// Mitsubishi GX Works2 project: Fx1NC-32MT-getfromInit   PLC: FX1N/FX1NC

PROGRAM MAIN
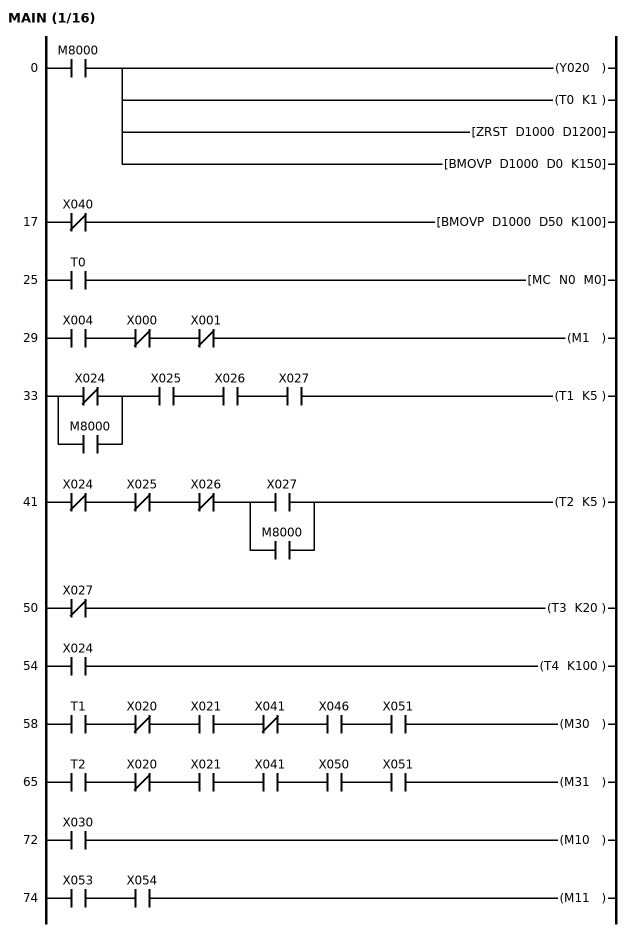
0     LD      M8000
      OUT     Y020
      OUT     T0 K1
      ZRST    D1000 D1200
      BMOVP   D1000 D0 K150
17    LDI     X040
      BMOVP   D1000 D50 K100
25    LD      T0
      MC      N0 M0
29    LD      X004
      ANI     X000
      ANI     X001
      OUT     M1
33    LDI     X024
      OR      M8000
      AND     X025
      AND     X026
      AND     X027
      OUT     T1 K5
41    LDI     X024
      ANI     X025
      ANI     X026
      LD      X027
      OR      M8000
      ANB
      OUT     T2 K5
50    LDI     X027
      OUT     T3 K20
54    LD      X024
      OUT     T4 K100
58    LD      T1
      ANI     X020
      AND     X021
      ANI     X041
      AND     X046
      AND     X051
      OUT     M30
65    LD      T2
      ANI     X020
      AND     X021
      AND     X041
      AND     X050
      AND     X051
      OUT     M31
72    LD      X030
      OUT     M10
74    LD      X053
      AND     X054
      OUT     M11
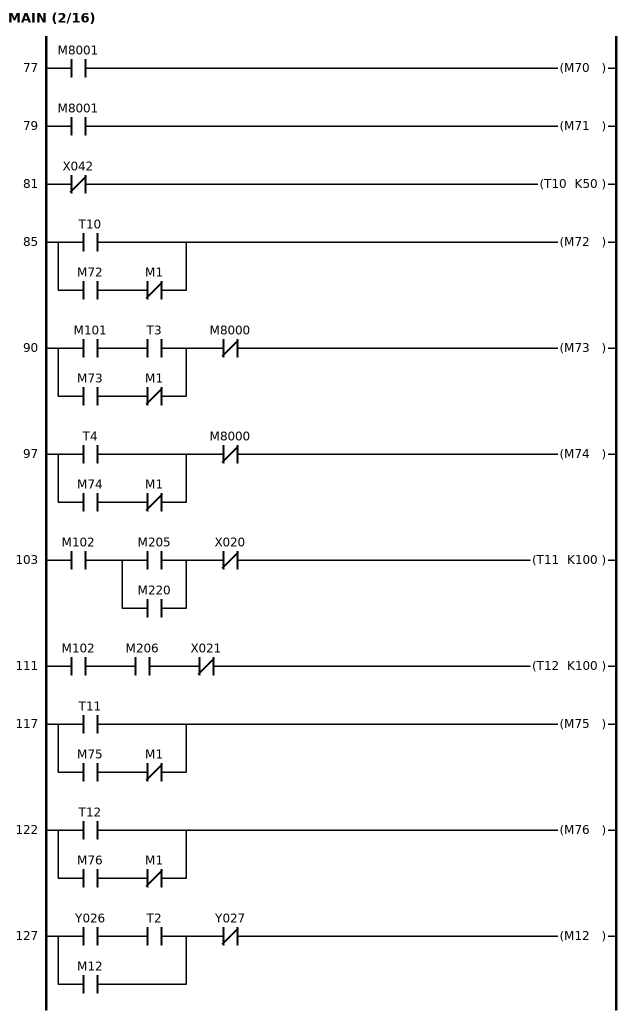
77    LD      M8001
      OUT     M70
79    LD      M8001
      OUT     M71
81    LDI     X042
      OUT     T10 K50
85    LD      T10
      LD      M72
      ANI     M1
      ORB
      OUT     M72
90    LD      M101
      AND     T3
      LD      M73
      ANI     M1
      ORB
      ANI     M8000
      OUT     M73
97    LD      T4
      LD      M74
      ANI     M1
      ORB
      ANI     M8000
      OUT     M74
103   LD      M102
      LD      M205
      OR      M220
      ANB
      ANI     X020
      OUT     T11 K100
111   LD      M102
      AND     M206
      ANI     X021
      OUT     T12 K100
117   LD      T11
      LD      M75
      ANI     M1
      ORB
      OUT     M75
122   LD      T12
      LD      M76
      ANI     M1
      ORB
      OUT     M76
127   LD      Y026
      AND     T2
      OR      M12
      ANI     Y027
      OUT     M12
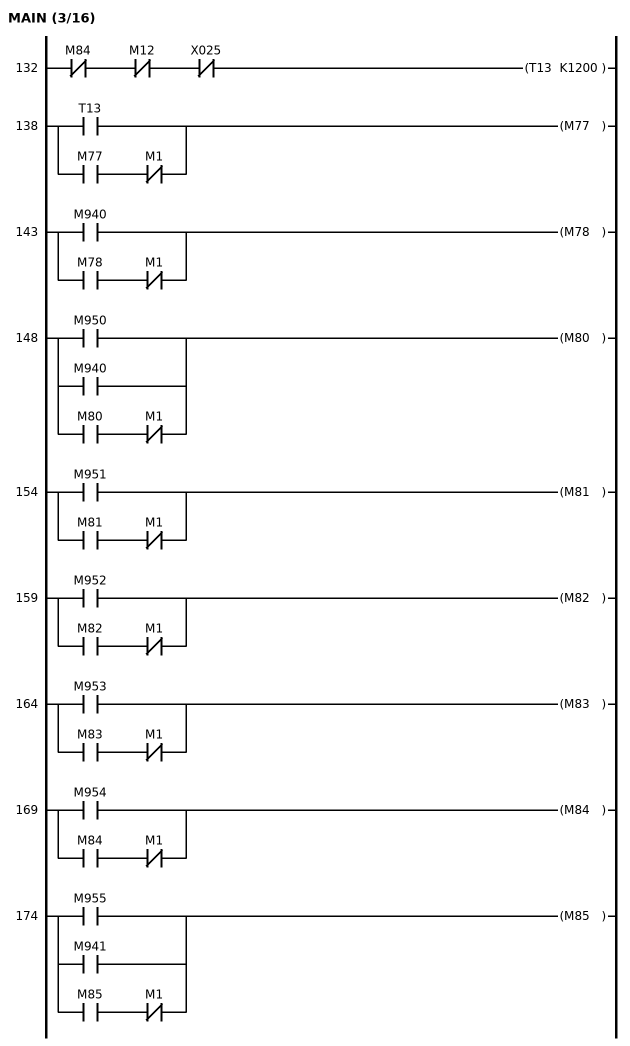
132   LDI     M84
      ANI     M12
      ANI     X025
      OUT     T13 K1200
138   LD      T13
      LD      M77
      ANI     M1
      ORB
      OUT     M77
143   LD      M940
      LD      M78
      ANI     M1
      ORB
      OUT     M78
148   LD      M950
      OR      M940
      LD      M80
      ANI     M1
      ORB
      OUT     M80
154   LD      M951
      LD      M81
      ANI     M1
      ORB
      OUT     M81
159   LD      M952
      LD      M82
      ANI     M1
      ORB
      OUT     M82
164   LD      M953
      LD      M83
      ANI     M1
      ORB
      OUT     M83
169   LD      M954
      LD      M84
      ANI     M1
      ORB
      OUT     M84
174   LD      M955
      OR      M941
      LD      M85
      ANI     M1
      ORB
      OUT     M85
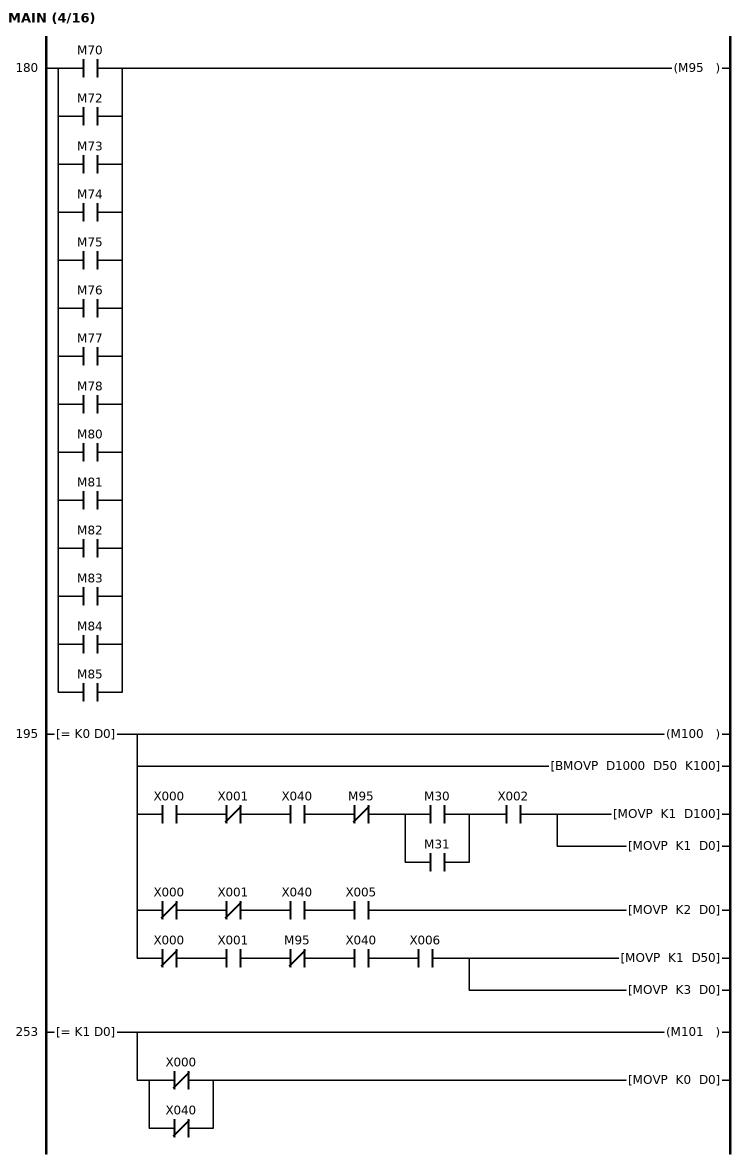
180   LD      M70
      OR      M72
      OR      M73
      OR      M74
      OR      M75
      OR      M76
      OR      M77
      OR      M78
      OR      M80
      OR      M81
      OR      M82
      OR      M83
      OR      M84
      OR      M85
      OUT     M95
195   LD=     K0 D0
      OUT     M100
      BMOVP   D1000 D50 K100
      MPS
      AND     X000
      ANI     X001
      AND     X040
      ANI     M95
      LD      M30
      OR      M31
      ANB
      AND     X002
      MOVP    K1 D100
      MOVP    K1 D0
      MRD
      ANI     X000
      ANI     X001
      AND     X040
      AND     X005
      MOVP    K2 D0
      MPP
      ANI     X000
      AND     X001
      ANI     M95
      AND     X040
      AND     X006
      MOVP    K1 D50
      MOVP    K3 D0
253   LD=     K1 D0
      OUT     M101
      LDI     X000
      ORI     X040
      ANB
      MOVP    K0 D0
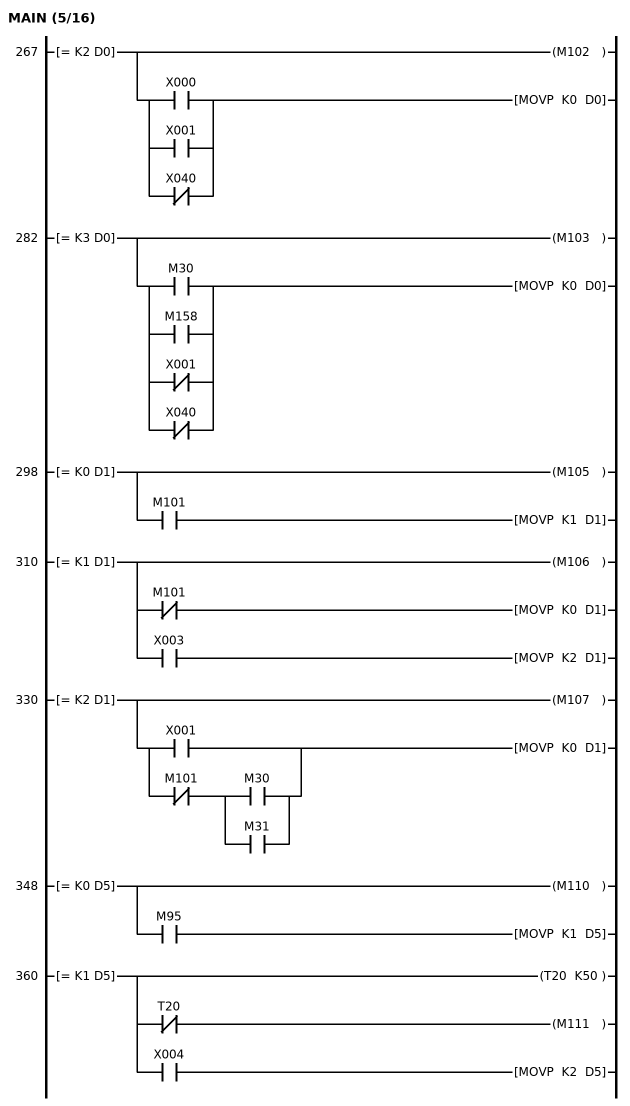
267   LD=     K2 D0
      OUT     M102
      LD      X000
      OR      X001
      ORI     X040
      ANB
      MOVP    K0 D0
282   LD=     K3 D0
      OUT     M103
      LD      M30
      OR      M158
      ORI     X001
      ORI     X040
      ANB
      MOVP    K0 D0
298   LD=     K0 D1
      OUT     M105
      AND     M101
      MOVP    K1 D1
310   LD=     K1 D1
      OUT     M106
      MPS
      ANI     M101
      MOVP    K0 D1
      MPP
      AND     X003
      MOVP    K2 D1
330   LD=     K2 D1
      OUT     M107
      LD      X001
      LDI     M101
      LD      M30
      OR      M31
      ANB
      ORB
      ANB
      MOVP    K0 D1
348   LD=     K0 D5
      OUT     M110
      AND     M95
      MOVP    K1 D5
360   LD=     K1 D5
      OUT     T20 K50
      MPS
      ANI     T20
      OUT     M111
      MPP
      AND     X004
      MOVP    K2 D5
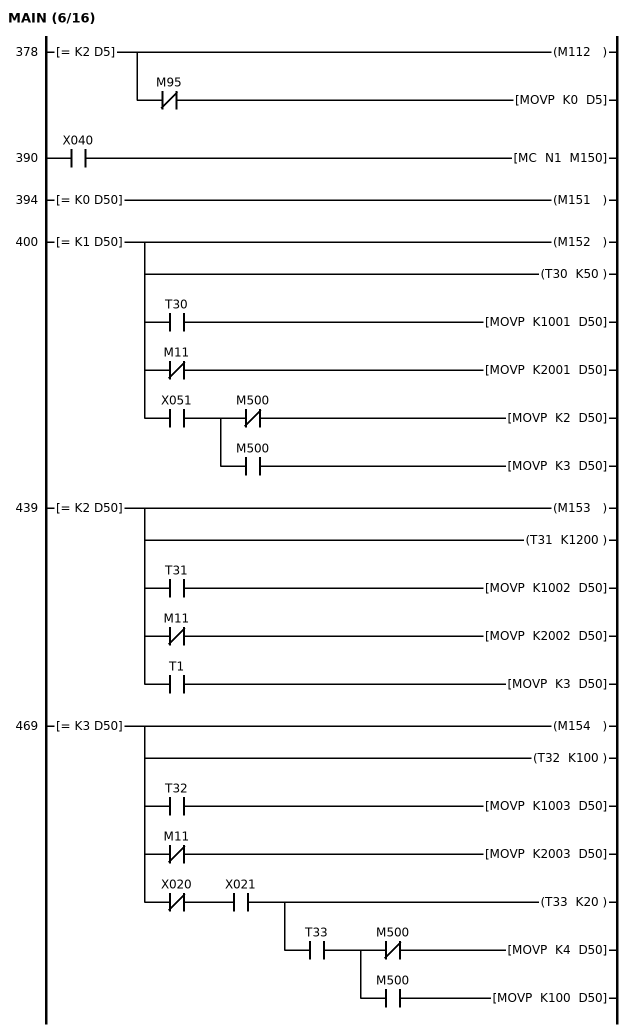
378   LD=     K2 D5
      OUT     M112
      ANI     M95
      MOVP    K0 D5
390   LD      X040
      MC      N1 M150
394   LD=     K0 D50
      OUT     M151
400   LD=     K1 D50
      OUT     M152
      OUT     T30 K50
      MPS
      AND     T30
      MOVP    K1001 D50
      MRD
      ANI     M11
      MOVP    K2001 D50
      MPP
      AND     X051
      MPS
      ANI     M500
      MOVP    K2 D50
      MPP
      AND     M500
      MOVP    K3 D50
439   LD=     K2 D50
      OUT     M153
      OUT     T31 K1200
      MPS
      AND     T31
      MOVP    K1002 D50
      MRD
      ANI     M11
      MOVP    K2002 D50
      MPP
      AND     T1
      MOVP    K3 D50
469   LD=     K3 D50
      OUT     M154
      OUT     T32 K100
      MPS
      AND     T32
      MOVP    K1003 D50
      MRD
      ANI     M11
      MOVP    K2003 D50
      MPP
      ANI     X020
      AND     X021
      OUT     T33 K20
      AND     T33
      MPS
      ANI     M500
      MOVP    K4 D50
      MPP
      AND     M500
      MOVP    K100 D50
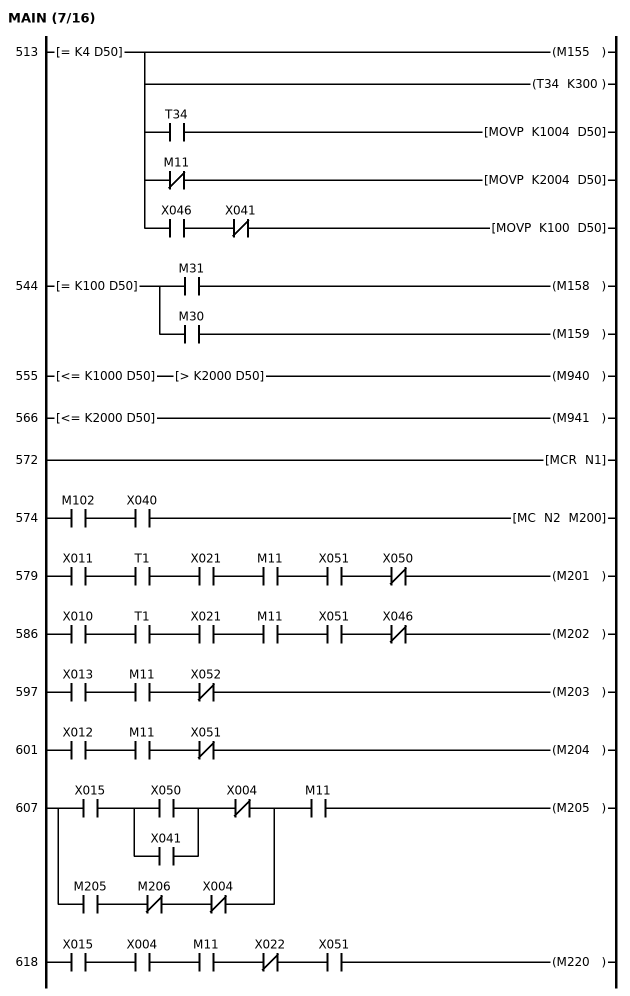
513   LD=     K4 D50
      OUT     M155
      OUT     T34 K300
      MPS
      AND     T34
      MOVP    K1004 D50
      MRD
      ANI     M11
      MOVP    K2004 D50
      MPP
      AND     X046
      ANI     X041
      MOVP    K100 D50
544   LD=     K100 D50
      MPS
      AND     M31
      OUT     M158
      MPP
      AND     M30
      OUT     M159
555   LD<=    K1000 D50
      AND>    K2000 D50
      OUT     M940
566   LD<=    K2000 D50
      OUT     M941
572   MCR     N1
574   LD      M102
      AND     X040
      MC      N2 M200
579   LD      X011
      AND     T1
      AND     X021
      AND     M11
      AND     X051
      ANI     X050
      OUT     M201
586   LD      X010
      AND     T1
      AND     X021
      AND     M11
      AND     X051
      ANI     X046
      OUT     M202
597   LD      X013
      AND     M11
      ANI     X052
      OUT     M203
601   LD      X012
      AND     M11
      ANI     X051
      OUT     M204
607   LD      X015
      LD      X050
      OR      X041
      ANB
      ANI     X004
      LD      M205
      ANI     M206
      ANI     X004
      ORB
      AND     M11
      OUT     M205
618   LD      X015
      AND     X004
      AND     M11
      ANI     X022
      AND     X051
      OUT     M220
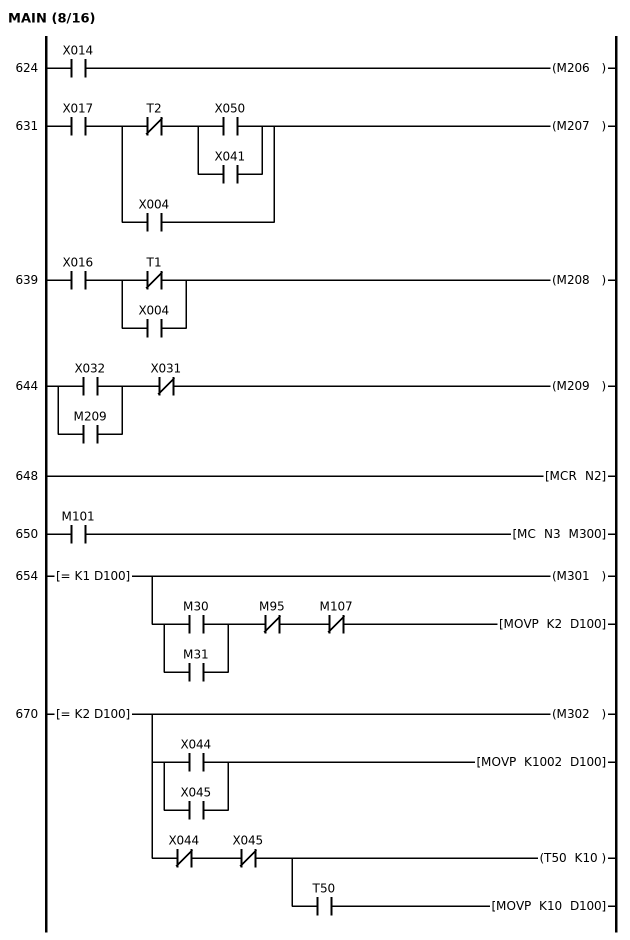
624   LD      X014
      OUT     M206
631   LD      X017
      LDI     T2
      LD      X050
      OR      X041
      ANB
      OR      X004
      ANB
      OUT     M207
639   LD      X016
      LDI     T1
      OR      X004
      ANB
      OUT     M208
644   LD      X032
      OR      M209
      ANI     X031
      OUT     M209
648   MCR     N2
650   LD      M101
      MC      N3 M300
654   LD=     K1 D100
      OUT     M301
      LD      M30
      OR      M31
      ANB
      ANI     M95
      ANI     M107
      MOVP    K2 D100
670   LD=     K2 D100
      OUT     M302
      MPS
      LD      X044
      OR      X045
      ANB
      MOVP    K1002 D100
      MPP
      ANI     X044
      ANI     X045
      OUT     T50 K10
      AND     T50
      MOVP    K10 D100
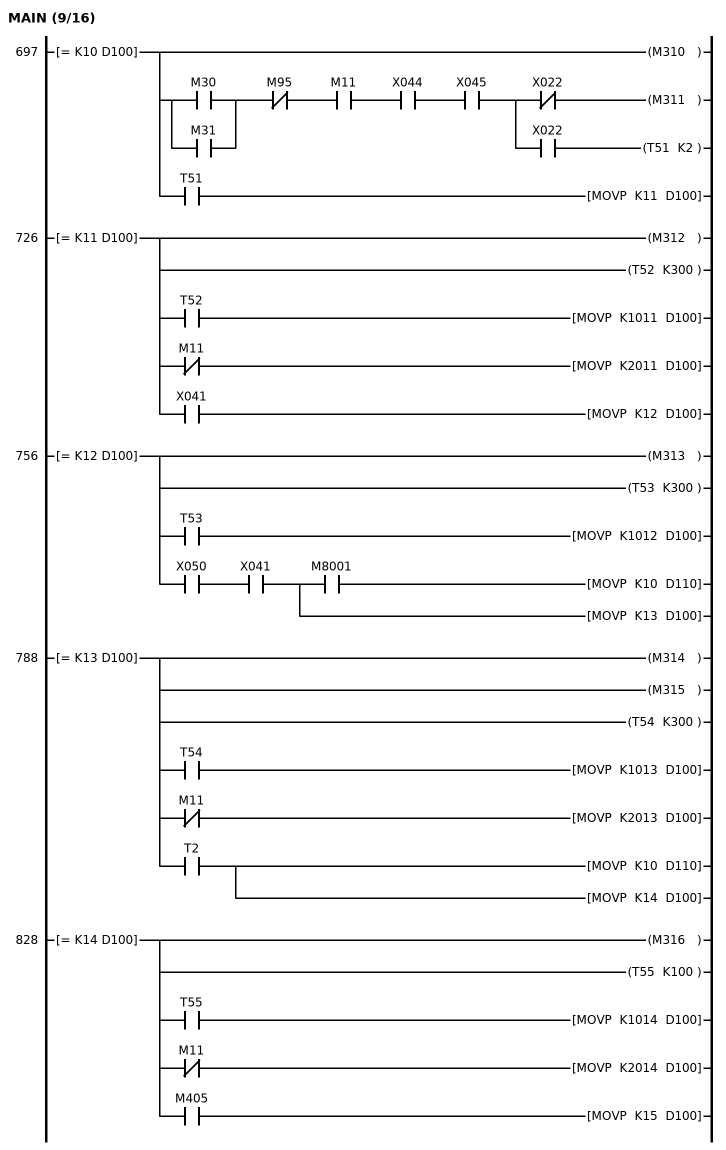
697   LD=     K10 D100
      OUT     M310
      MPS
      LD      M30
      OR      M31
      ANB
      ANI     M95
      AND     M11
      AND     X044
      AND     X045
      MPS
      ANI     X022
      OUT     M311
      MPP
      AND     X022
      OUT     T51 K2
      MPP
      AND     T51
      MOVP    K11 D100
726   LD=     K11 D100
      OUT     M312
      OUT     T52 K300
      MPS
      AND     T52
      MOVP    K1011 D100
      MRD
      ANI     M11
      MOVP    K2011 D100
      MPP
      AND     X041
      MOVP    K12 D100
756   LD=     K12 D100
      OUT     M313
      OUT     T53 K300
      MPS
      AND     T53
      MOVP    K1012 D100
      MPP
      AND     X050
      AND     X041
      MPS
      AND     M8001
      MOVP    K10 D110
      MPP
      MOVP    K13 D100
788   LD=     K13 D100
      OUT     M314
      OUT     M315
      OUT     T54 K300
      MPS
      AND     T54
      MOVP    K1013 D100
      MRD
      ANI     M11
      MOVP    K2013 D100
      MPP
      AND     T2
      MOVP    K10 D110
      MOVP    K14 D100
828   LD=     K14 D100
      OUT     M316
      OUT     T55 K100
      MPS
      AND     T55
      MOVP    K1014 D100
      MRD
      ANI     M11
      MOVP    K2014 D100
      MPP
      AND     M405
      MOVP    K15 D100
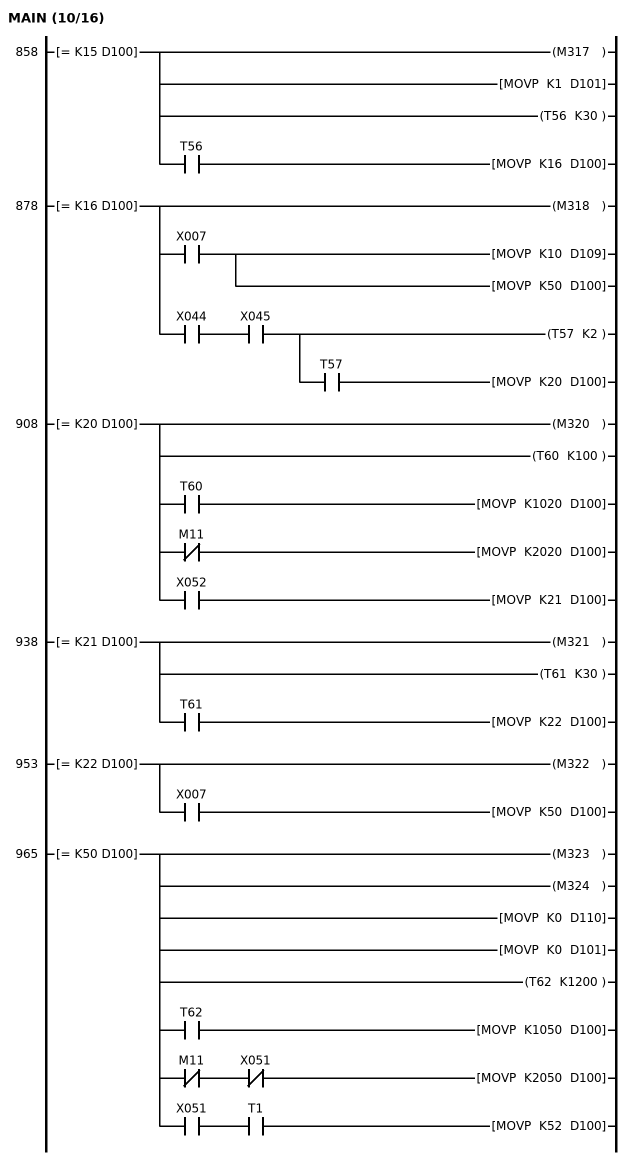
858   LD=     K15 D100
      OUT     M317
      MOVP    K1 D101
      OUT     T56 K30
      AND     T56
      MOVP    K16 D100
878   LD=     K16 D100
      OUT     M318
      MPS
      AND     X007
      MOVP    K10 D109
      MOVP    K50 D100
      MPP
      AND     X044
      AND     X045
      OUT     T57 K2
      AND     T57
      MOVP    K20 D100
908   LD=     K20 D100
      OUT     M320
      OUT     T60 K100
      MPS
      AND     T60
      MOVP    K1020 D100
      MRD
      ANI     M11
      MOVP    K2020 D100
      MPP
      AND     X052
      MOVP    K21 D100
938   LD=     K21 D100
      OUT     M321
      OUT     T61 K30
      AND     T61
      MOVP    K22 D100
953   LD=     K22 D100
      OUT     M322
      AND     X007
      MOVP    K50 D100
965   LD=     K50 D100
      OUT     M323
      OUT     M324
      MOVP    K0 D110
      MOVP    K0 D101
      OUT     T62 K1200
      MPS
      AND     T62
      MOVP    K1050 D100
      MRD
      ANI     M11
      ANI     X051
      MOVP    K2050 D100
      MPP
      AND     X051
      AND     T1
      MOVP    K52 D100
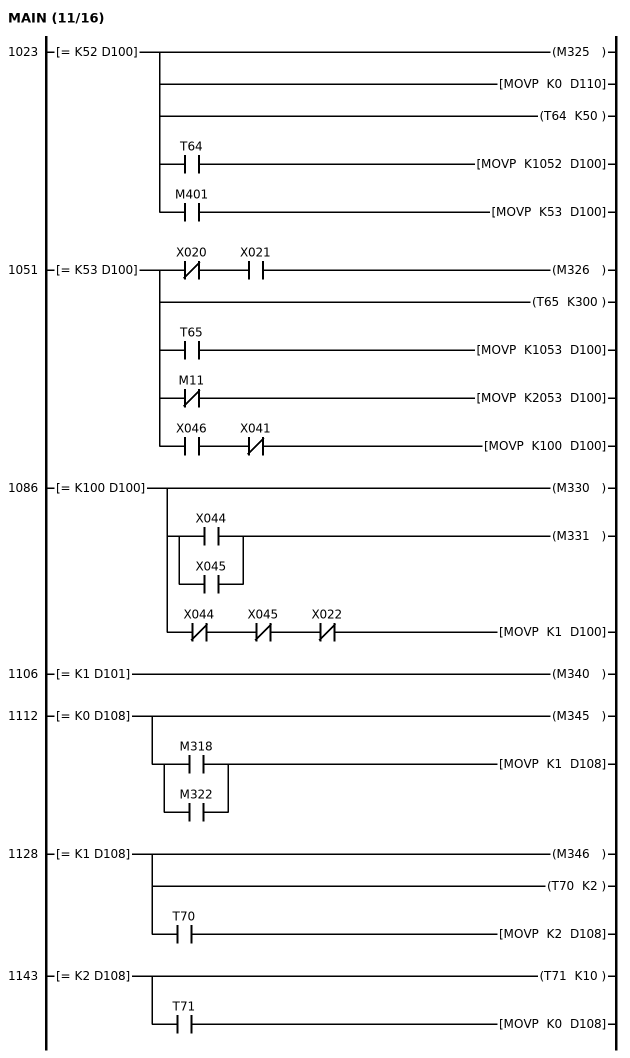
1023  LD=     K52 D100
      OUT     M325
      MOVP    K0 D110
      OUT     T64 K50
      MPS
      AND     T64
      MOVP    K1052 D100
      MPP
      AND     M401
      MOVP    K53 D100
1051  LD=     K53 D100
      MPS
      ANI     X020
      AND     X021
      OUT     M326
      MPP
      OUT     T65 K300
      MPS
      AND     T65
      MOVP    K1053 D100
      MRD
      ANI     M11
      MOVP    K2053 D100
      MPP
      AND     X046
      ANI     X041
      MOVP    K100 D100
1086  LD=     K100 D100
      OUT     M330
      MPS
      LD      X044
      OR      X045
      ANB
      OUT     M331
      MPP
      ANI     X044
      ANI     X045
      ANI     X022
      MOVP    K1 D100
1106  LD=     K1 D101
      OUT     M340
1112  LD=     K0 D108
      OUT     M345
      LD      M318
      OR      M322
      ANB
      MOVP    K1 D108
1128  LD=     K1 D108
      OUT     M346
      OUT     T70 K2
      AND     T70
      MOVP    K2 D108
1143  LD=     K2 D108
      OUT     T71 K10
      AND     T71
      MOVP    K0 D108
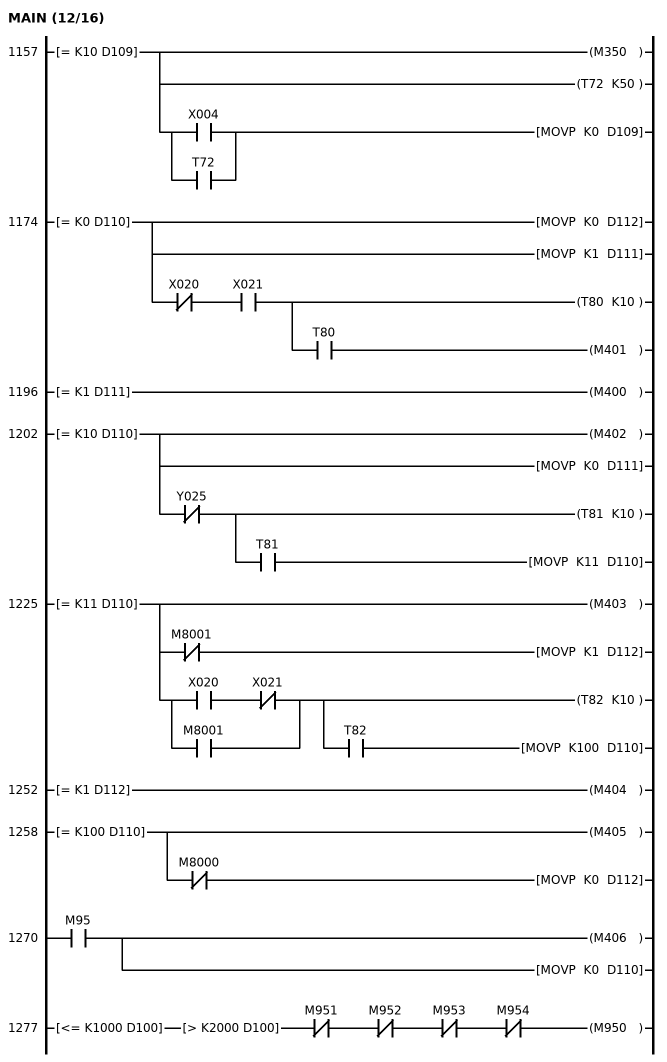
1157  LD=     K10 D109
      OUT     M350
      OUT     T72 K50
      LD      X004
      OR      T72
      ANB
      MOVP    K0 D109
1174  LD=     K0 D110
      MOVP    K0 D112
      MOVP    K1 D111
      ANI     X020
      AND     X021
      OUT     T80 K10
      AND     T80
      OUT     M401
1196  LD=     K1 D111
      OUT     M400
1202  LD=     K10 D110
      OUT     M402
      MOVP    K0 D111
      ANI     Y025
      OUT     T81 K10
      AND     T81
      MOVP    K11 D110
1225  LD=     K11 D110
      OUT     M403
      MPS
      ANI     M8001
      MOVP    K1 D112
      MPP
      LD      X020
      ANI     X021
      OR      M8001
      ANB
      OUT     T82 K10
      AND     T82
      MOVP    K100 D110
1252  LD=     K1 D112
      OUT     M404
1258  LD=     K100 D110
      OUT     M405
      ANI     M8000
      MOVP    K0 D112
1270  LD      M95
      OUT     M406
      MOVP    K0 D110
1277  LD<=    K1000 D100
      AND>    K2000 D100
      ANI     M951
      ANI     M952
      ANI     M953
      ANI     M954
      OUT     M950
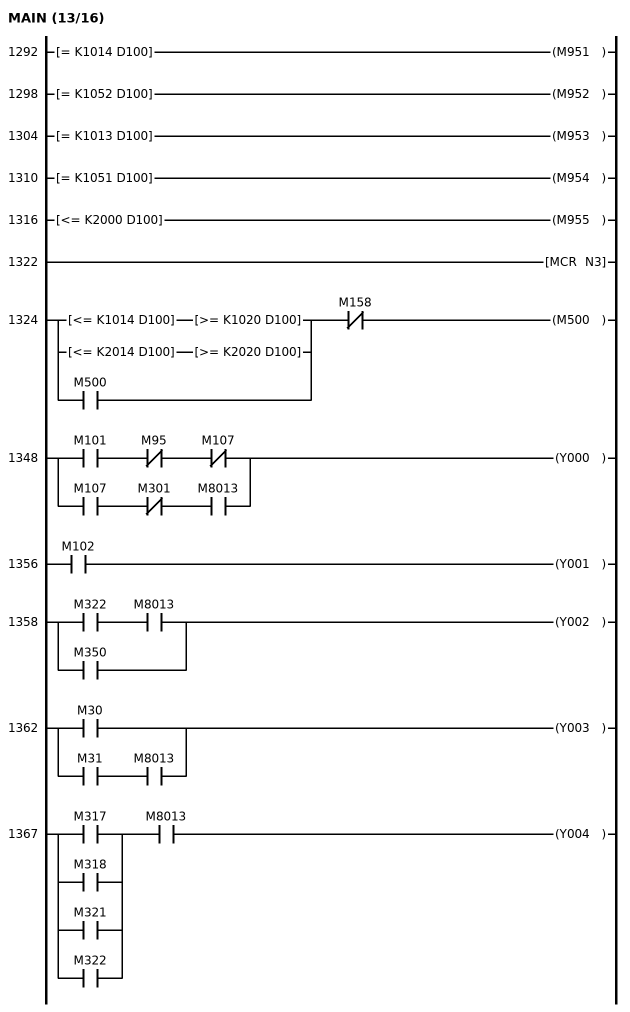
1292  LD=     K1014 D100
      OUT     M951
1298  LD=     K1052 D100
      OUT     M952
1304  LD=     K1013 D100
      OUT     M953
1310  LD=     K1051 D100
      OUT     M954
1316  LD<=    K2000 D100
      OUT     M955
1322  MCR     N3
1324  LD<=    K1014 D100
      AND>=   K1020 D100
      LD<=    K2014 D100
      AND>=   K2020 D100
      ORB
      OR      M500
      ANI     M158
      OUT     M500
1348  LD      M101
      ANI     M95
      ANI     M107
      LD      M107
      ANI     M301
      AND     M8013
      ORB
      OUT     Y000
1356  LD      M102
      OUT     Y001
1358  LD      M322
      AND     M8013
      OR      M350
      OUT     Y002
1362  LD      M30
      LD      M31
      AND     M8013
      ORB
      OUT     Y003
1367  LD      M317
      OR      M318
      OR      M321
      OR      M322
      AND     M8013
      OUT     Y004
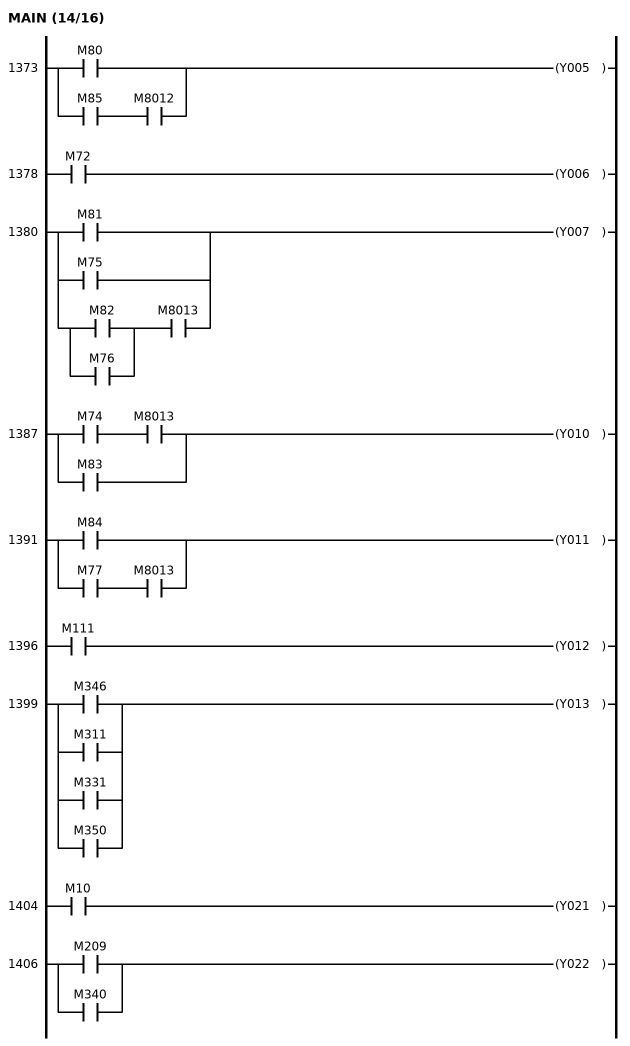
1373  LD      M80
      LD      M85
      AND     M8012
      ORB
      OUT     Y005
1378  LD      M72
      OUT     Y006
1380  LD      M81
      OR      M75
      LD      M82
      OR      M76
      AND     M8013
      ORB
      OUT     Y007
1387  LD      M74
      AND     M8013
      OR      M83
      OUT     Y010
1391  LD      M84
      LD      M77
      AND     M8013
      ORB
      OUT     Y011
1396  LD      M111
      OUT     Y012
1399  LD      M346
      OR      M311
      OR      M331
      OR      M350
      OUT     Y013
1404  LD      M10
      OUT     Y021
1406  LD      M209
      OR      M340
      OUT     Y022
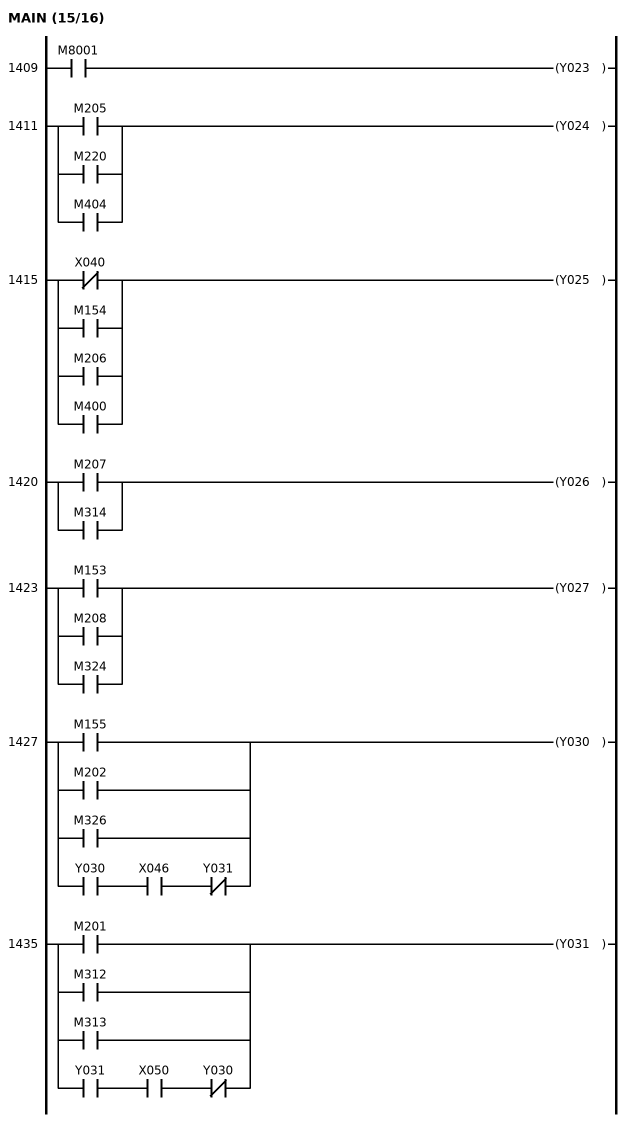
1409  LD      M8001
      OUT     Y023
1411  LD      M205
      OR      M220
      OR      M404
      OUT     Y024
1415  LDI     X040
      OR      M154
      OR      M206
      OR      M400
      OUT     Y025
1420  LD      M207
      OR      M314
      OUT     Y026
1423  LD      M153
      OR      M208
      OR      M324
      OUT     Y027
1427  LD      M155
      OR      M202
      OR      M326
      LD      Y030
      AND     X046
      ANI     Y031
      ORB
      OUT     Y030
1435  LD      M201
      OR      M312
      OR      M313
      LD      Y031
      AND     X050
      ANI     Y030
      ORB
      OUT     Y031
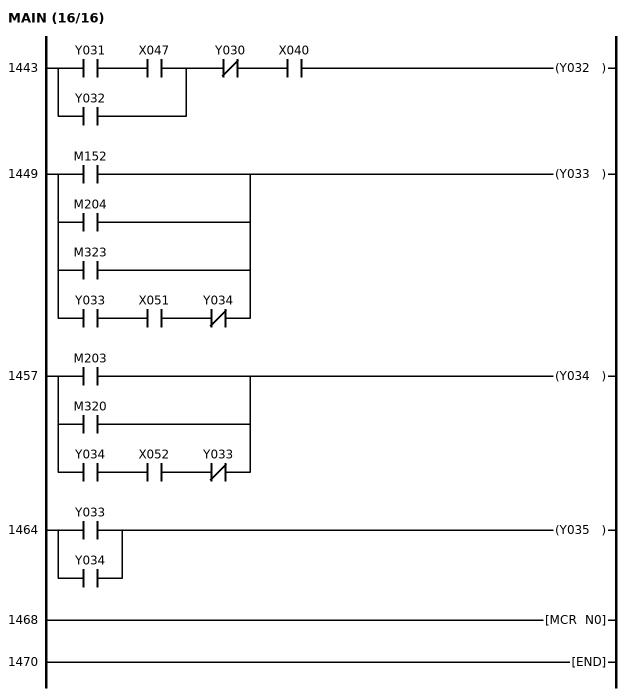
1443  LD      Y031
      AND     X047
      OR      Y032
      ANI     Y030
      AND     X040
      OUT     Y032
1449  LD      M152
      OR      M204
      OR      M323
      LD      Y033
      AND     X051
      ANI     Y034
      ORB
      OUT     Y033
1457  LD      M203
      OR      M320
      LD      Y034
      AND     X052
      ANI     Y033
      ORB
      OUT     Y034
1464  LD      Y033
      OR      Y034
      OUT     Y035
1468  MCR     N0
1470  END
END_PROGRAM
